// Mitsubishi GX Works2 project: MyProject-PLC   PLC: FX3U/FX3UC

PROGRAM MAIN
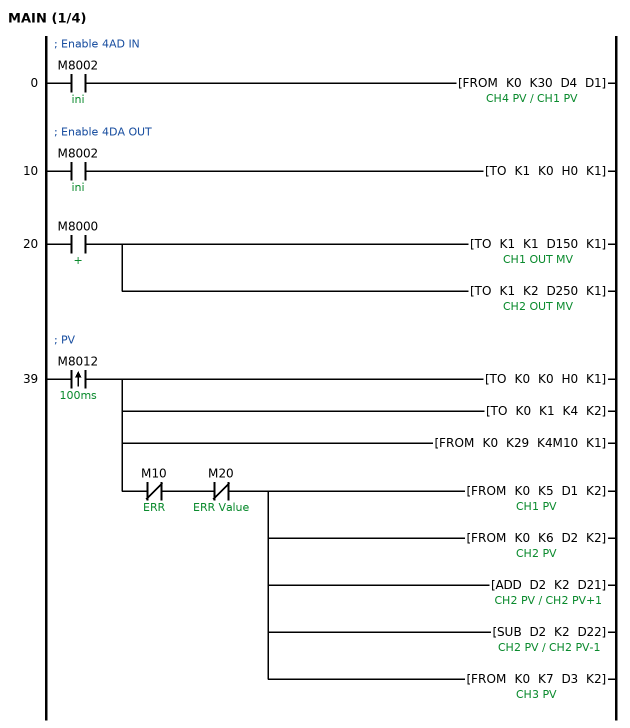
; Enable 4AD IN
0     LD      M8002  ; ini
      FROM    K0 K30 D4 D1  ; CH4 PV / CH1 PV
; Enable 4DA OUT
10    LD      M8002  ; ini
      TO      K1 K0 H0 K1
20    LD      M8000  ; +
      TO      K1 K1 D150 K1  ; CH1 OUT MV
      TO      K1 K2 D250 K1  ; CH2 OUT MV
; PV
39    LDP     M8012  ; 100ms
      TO      K0 K0 H0 K1
      TO      K0 K1 K4 K2
      FROM    K0 K29 K4M10 K1  ; ERR
      ANI     M10  ; ERR
      ANI     M20  ; ERR Value
      FROM    K0 K5 D1 K2
      FROM    K0 K6 D2 K2  ; CH2 PV
      ADD     D2 K2 D21  ; CH2 PV+1
      SUB     D2 K2 D22  ; CH2 PV-1
      FROM    K0 K7 D3 K2  ; CH3 PV
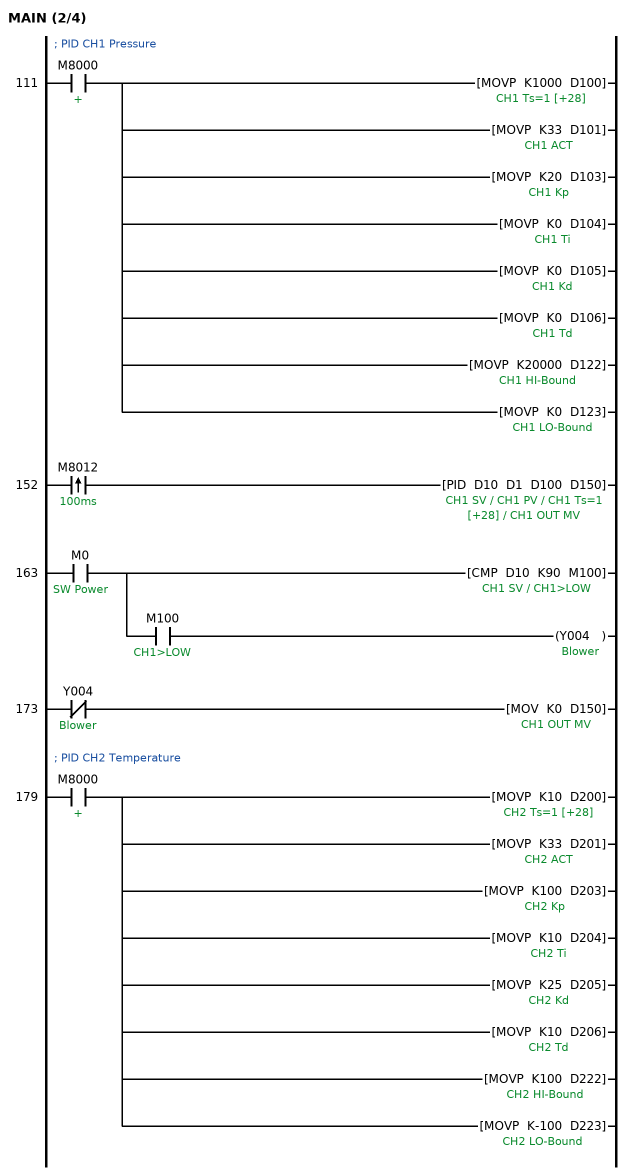
; PID CH1 Pressure
111   LD      M8000  ; +
      MOVP    K1000 D100  ; CH1 Ts=1 [+28]
      MOVP    K33 D101  ; CH1 ACT
      MOVP    K20 D103  ; CH1 Kp
      MOVP    K0 D104  ; CH1 Ti
      MOVP    K0 D105  ; CH1 Kd
      MOVP    K0 D106  ; CH1 Td
      MOVP    K20000 D122  ; CH1 HI-Bound
      MOVP    K0 D123  ; CH1 LO-Bound
152   LDP     M8012  ; 100ms
      PID     D10 D1 D100 D150  ; CH1 SV
163   LD      M0  ; SW Power
      CMP     D10 K90 M100  ; CH1>LOW
      AND     M100  ; CH1>LOW
      OUT     Y004  ; Blower
173   LDI     Y004  ; Blower
      MOV     K0 D150
; PID CH2 Temperature
179   LD      M8000  ; +
      MOVP    K10 D200  ; CH2 Ts=1 [+28]
      MOVP    K33 D201  ; CH2 ACT
      MOVP    K100 D203  ; CH2 Kp
      MOVP    K10 D204  ; CH2 Ti
      MOVP    K25 D205  ; CH2 Kd
      MOVP    K10 D206  ; CH2 Td
      MOVP    K100 D222  ; CH2 HI-Bound
      MOVP    K-100 D223  ; CH2 LO-Bound
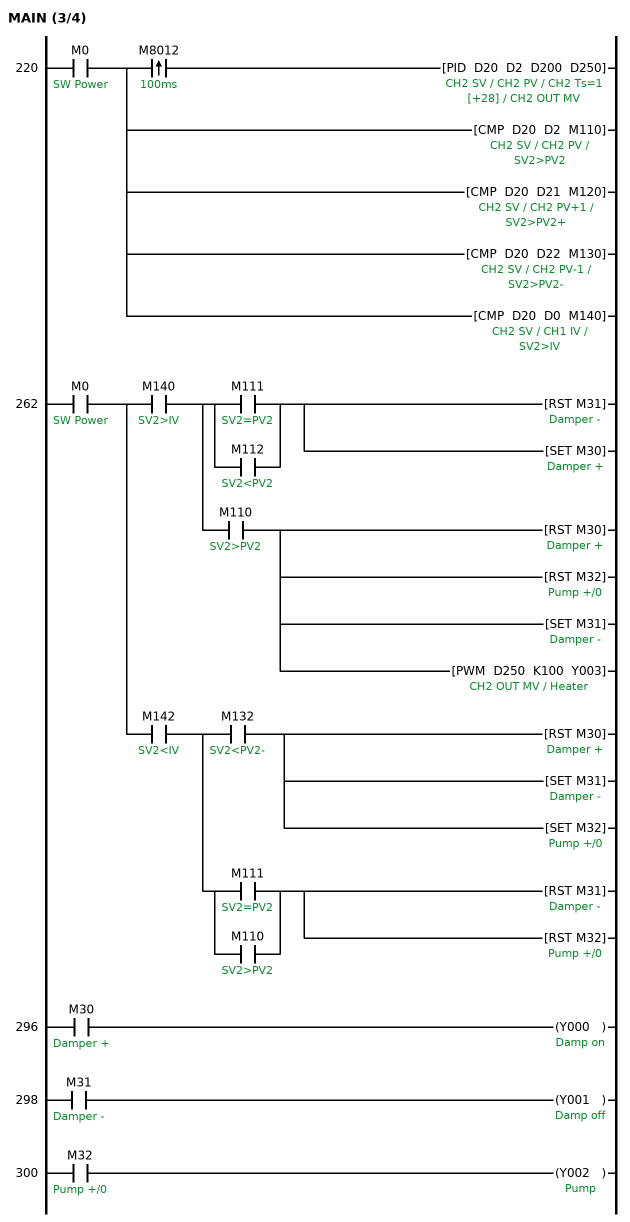
220   LD      M0  ; SW Power
      MPS
      ANDP    M8012  ; 100ms
      PID     D20 D2 D200 D250  ; CH2 SV
      MPP
      CMP     D20 D2 M110  ; SV2>PV2
      CMP     D20 D21 M120  ; SV2>PV2+
      CMP     D20 D22 M130  ; SV2>PV2-
      CMP     D20 D0 M140  ; CH1 IV / SV2>IV
262   LD      M0  ; SW Power
      MPS
      AND     M140  ; SV2>IV
      MPS
      LD      M111  ; SV2=PV2
      OR      M112  ; SV2<PV2
      ANB
      RST     M31  ; Damper -
      SET     M30  ; Damper +
      MPP
      AND     M110  ; SV2>PV2
      RST     M30  ; Damper +
      RST     M32  ; Pump +/0
      SET     M31  ; Damper -
      PWM     D250 K100 Y003  ; Heater
      MPP
      AND     M142  ; SV2<IV
      MPS
      AND     M132  ; SV2<PV2-
      RST     M30  ; Damper +
      SET     M31  ; Damper -
      SET     M32  ; Pump +/0
      MPP
      LD      M111  ; SV2=PV2
      OR      M110  ; SV2>PV2
      ANB
      RST     M31  ; Damper -
      RST     M32  ; Pump +/0
296   LD      M30  ; Damper +
      OUT     Y000  ; Damp on
298   LD      M31  ; Damper -
      OUT     Y001  ; Damp off
300   LD      M32  ; Pump +/0
      OUT     Y002  ; Pump
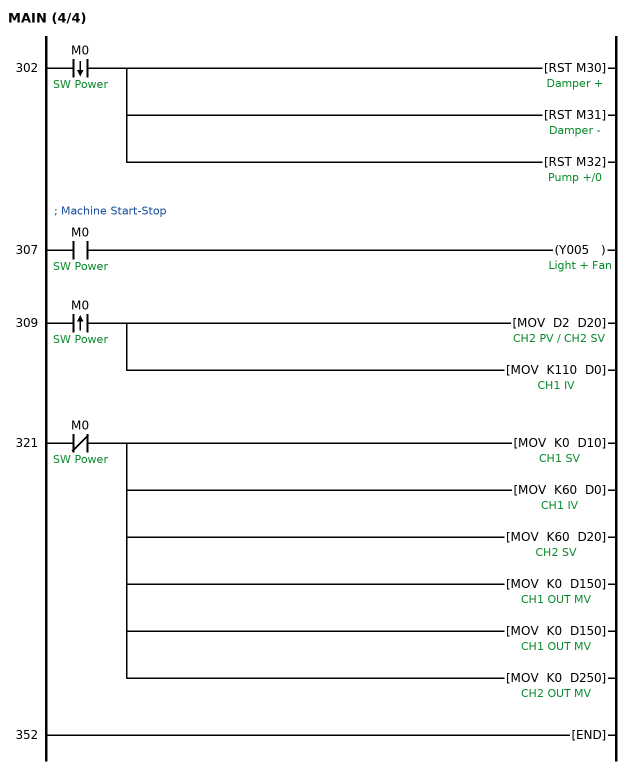
302   LDF     M0  ; SW Power
      RST     M30  ; Damper +
      RST     M31  ; Damper -
      RST     M32  ; Pump +/0
; Machine Start-Stop
307   LD      M0  ; SW Power
      OUT     Y005  ; Light + Fan
309   LDP     M0  ; SW Power
      MOV     D2 D20
      MOV     K110 D0
321   LDI     M0  ; SW Power
      MOV     K0 D10
      MOV     K60 D0
      MOV     K60 D20
      MOV     K0 D150
      MOV     K0 D150
      MOV     K0 D250
352   END
END_PROGRAM

// device comments not shown above
M1  ; SW OPC SetSV
M101  ; CH1=LOW
M102  ; CH1<LOW
M121  ; SV2=PV2+
M122  ; SV2<PV2+
M131  ; SV2=PV2-
M141  ; SV2=IV
M555  ; comment
M1000  ; Test On-Off
M2000  ; Comment Off
